// TIA Portal V21 export
FUNCTION "ModeSelect" : Void   // FC7, LAD
{ S7_Optimized_Access := 'TRUE' }
// stored: AutoNumber false, SetENOAutomatically false
BEGIN

REGION Network 1: ****************************MV3000_Enable *****************************
END_REGION

REGION Network 2: "ModeDb".MV3000.Mode.ManualMode.Enable
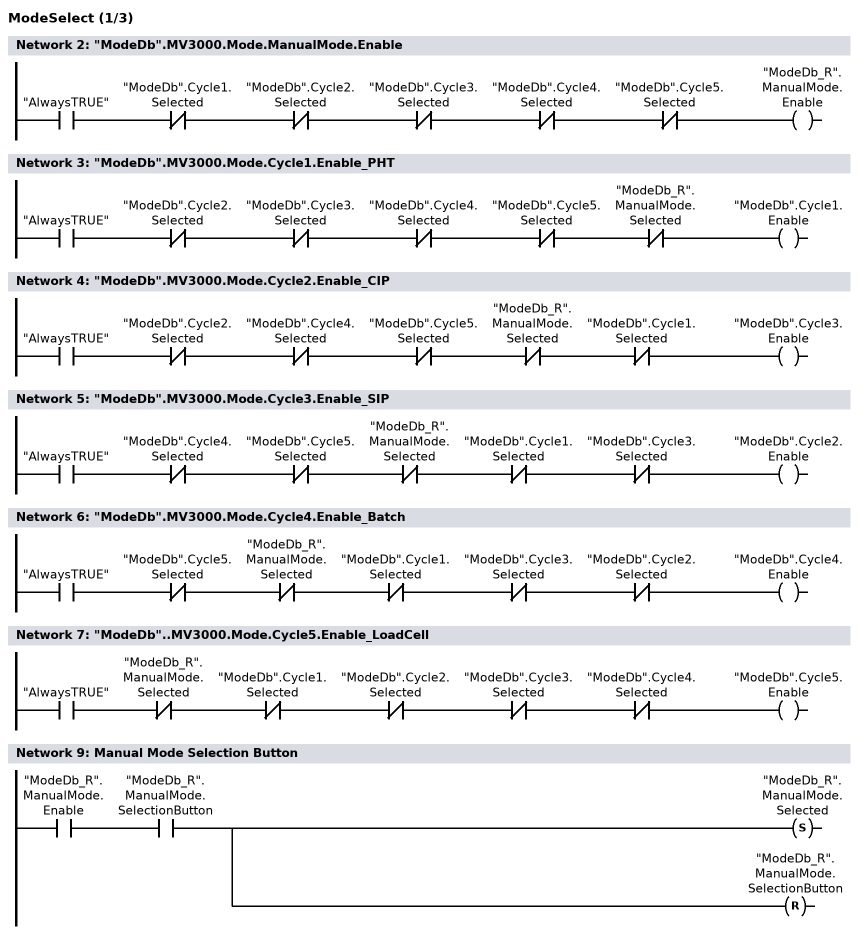
   RUNG wire#powerrail
      Contact( "AlwaysTRUE" )
      I_Contact( "ModeDb".Cycle1.Selected )
      I_Contact( "ModeDb".Cycle2.Selected )
      I_Contact( "ModeDb".Cycle3.Selected )
      I_Contact( "ModeDb".Cycle4.Selected )
      I_Contact( "ModeDb".Cycle5.Selected )
      Coil( "ModeDb_R".ManualMode.Enable )
   END_RUNG
   // the same network as SCL:
   "ModeDb_R".ManualMode.Enable := "AlwaysTRUE" AND NOT "ModeDb".Cycle1.Selected AND NOT "ModeDb".Cycle2.Selected AND NOT "ModeDb".Cycle3.Selected AND NOT "ModeDb".Cycle4.Selected AND NOT "ModeDb".Cycle5.Selected;
END_REGION

REGION Network 3: "ModeDb".MV3000.Mode.Cycle1.Enable_PHT
   RUNG wire#powerrail
      Contact( "AlwaysTRUE" )
      I_Contact( "ModeDb".Cycle2.Selected )
      I_Contact( "ModeDb".Cycle3.Selected )
      I_Contact( "ModeDb".Cycle4.Selected )
      I_Contact( "ModeDb".Cycle5.Selected )
      I_Contact( "ModeDb_R".ManualMode.Selected )
      Coil( "ModeDb".Cycle1.Enable )
   END_RUNG
   // the same network as SCL:
   "ModeDb".Cycle1.Enable := "AlwaysTRUE" AND NOT "ModeDb".Cycle2.Selected AND NOT "ModeDb".Cycle3.Selected AND NOT "ModeDb".Cycle4.Selected AND NOT "ModeDb".Cycle5.Selected AND NOT "ModeDb_R".ManualMode.Selected;
END_REGION

REGION Network 4: "ModeDb".MV3000.Mode.Cycle2.Enable_CIP
   RUNG wire#powerrail
      Contact( "AlwaysTRUE" )
      I_Contact( "ModeDb".Cycle2.Selected )
      I_Contact( "ModeDb".Cycle4.Selected )
      I_Contact( "ModeDb".Cycle5.Selected )
      I_Contact( "ModeDb_R".ManualMode.Selected )
      I_Contact( "ModeDb".Cycle1.Selected )
      Coil( "ModeDb".Cycle3.Enable )
   END_RUNG
   // the same network as SCL:
   "ModeDb".Cycle3.Enable := "AlwaysTRUE" AND NOT "ModeDb".Cycle2.Selected AND NOT "ModeDb".Cycle4.Selected AND NOT "ModeDb".Cycle5.Selected AND NOT "ModeDb_R".ManualMode.Selected AND NOT "ModeDb".Cycle1.Selected;
END_REGION

REGION Network 5: "ModeDb".MV3000.Mode.Cycle3.Enable_SIP
   RUNG wire#powerrail
      Contact( "AlwaysTRUE" )
      I_Contact( "ModeDb".Cycle4.Selected )
      I_Contact( "ModeDb".Cycle5.Selected )
      I_Contact( "ModeDb_R".ManualMode.Selected )
      I_Contact( "ModeDb".Cycle1.Selected )
      I_Contact( "ModeDb".Cycle3.Selected )
      Coil( "ModeDb".Cycle2.Enable )
   END_RUNG
   // the same network as SCL:
   "ModeDb".Cycle2.Enable := "AlwaysTRUE" AND NOT "ModeDb".Cycle4.Selected AND NOT "ModeDb".Cycle5.Selected AND NOT "ModeDb_R".ManualMode.Selected AND NOT "ModeDb".Cycle1.Selected AND NOT "ModeDb".Cycle3.Selected;
END_REGION

REGION Network 6: "ModeDb".MV3000.Mode.Cycle4.Enable_Batch
   RUNG wire#powerrail
      Contact( "AlwaysTRUE" )
      I_Contact( "ModeDb".Cycle5.Selected )
      I_Contact( "ModeDb_R".ManualMode.Selected )
      I_Contact( "ModeDb".Cycle1.Selected )
      I_Contact( "ModeDb".Cycle3.Selected )
      I_Contact( "ModeDb".Cycle2.Selected )
      Coil( "ModeDb".Cycle4.Enable )
   END_RUNG
   // the same network as SCL:
   "ModeDb".Cycle4.Enable := "AlwaysTRUE" AND NOT "ModeDb".Cycle5.Selected AND NOT "ModeDb_R".ManualMode.Selected AND NOT "ModeDb".Cycle1.Selected AND NOT "ModeDb".Cycle3.Selected AND NOT "ModeDb".Cycle2.Selected;
END_REGION

REGION Network 7: "ModeDb"..MV3000.Mode.Cycle5.Enable_LoadCell
   RUNG wire#powerrail
      Contact( "AlwaysTRUE" )
      I_Contact( "ModeDb_R".ManualMode.Selected )
      I_Contact( "ModeDb".Cycle1.Selected )
      I_Contact( "ModeDb".Cycle2.Selected )
      I_Contact( "ModeDb".Cycle3.Selected )
      I_Contact( "ModeDb".Cycle4.Selected )
      Coil( "ModeDb".Cycle5.Enable )
   END_RUNG
   // the same network as SCL:
   "ModeDb".Cycle5.Enable := "AlwaysTRUE" AND NOT "ModeDb_R".ManualMode.Selected AND NOT "ModeDb".Cycle1.Selected AND NOT "ModeDb".Cycle2.Selected AND NOT "ModeDb".Cycle3.Selected AND NOT "ModeDb".Cycle4.Selected;
END_REGION

REGION Network 8: ------------------------------------------------- SELECTION BUTTON -------------------------------------------------
END_REGION

REGION Network 9: Manual Mode Selection Button
   RUNG wire#powerrail
      Contact( "ModeDb_R".ManualMode.Enable )
      Contact( "ModeDb_R".ManualMode.SelectionButton )
      wire#w1
      S_Coil( "ModeDb_R".ManualMode.Selected )
   END_RUNG
   RUNG wire#w1
      R_Coil( "ModeDb_R".ManualMode.SelectionButton )
   END_RUNG
   // the same network as SCL:
   IF "ModeDb_R".ManualMode.Enable AND "ModeDb_R".ManualMode.SelectionButton THEN
       "ModeDb_R".ManualMode.Selected := TRUE;
       "ModeDb_R".ManualMode.SelectionButton := FALSE;
   END_IF;
END_REGION

REGION Network 10: __________________________ VESSEL STATUS__________________________
END_REGION

REGION Network 11: "HmiTags".Cv200VesselStatus
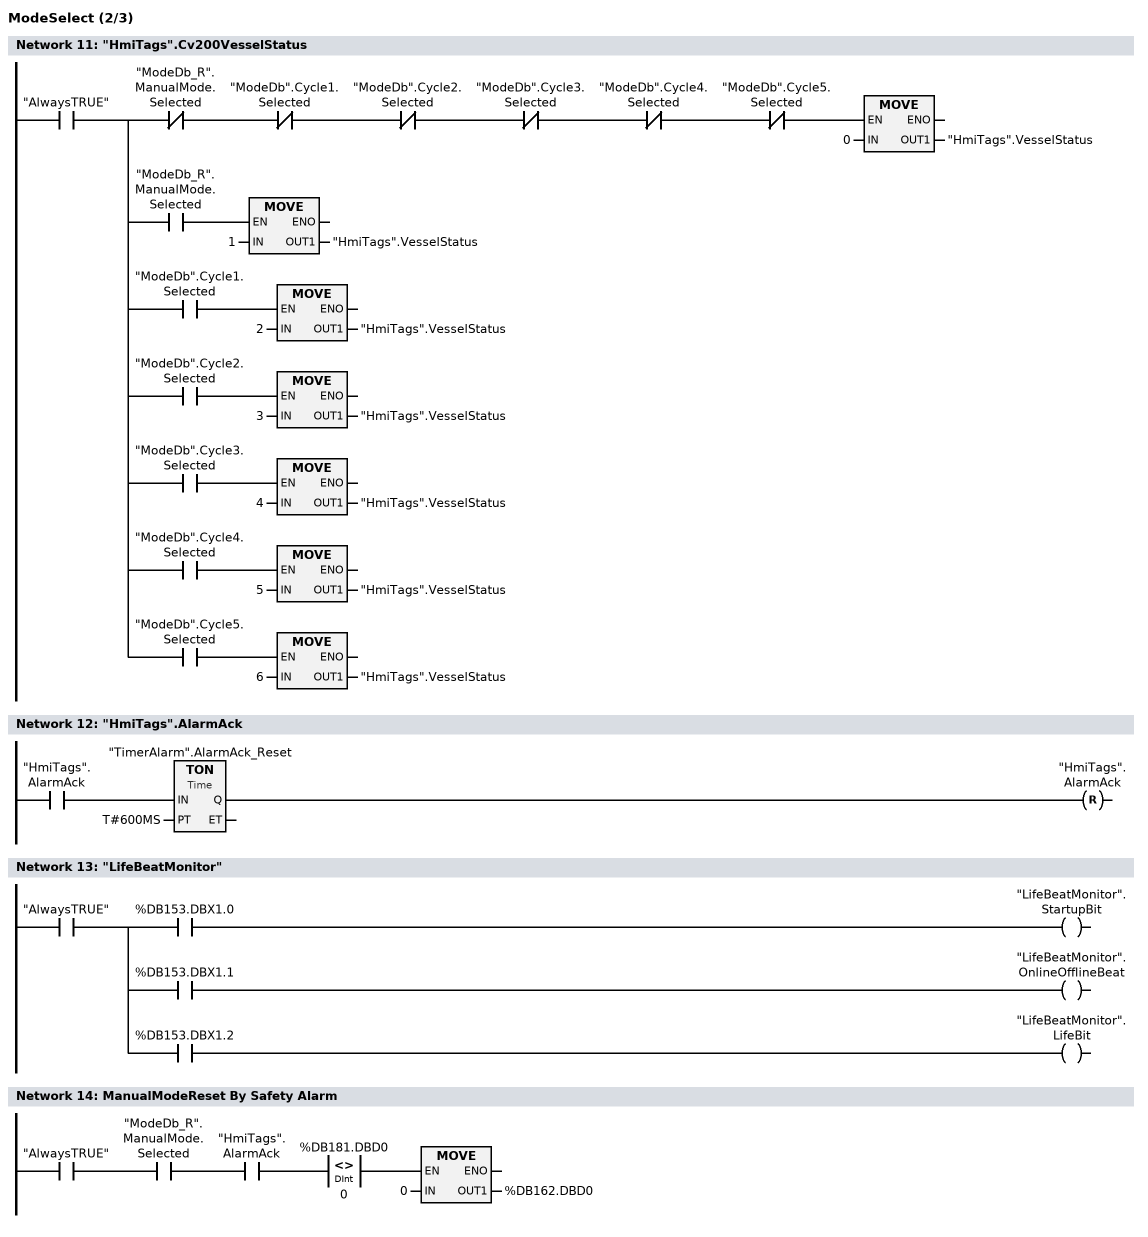
   RUNG wire#powerrail
      Contact( "AlwaysTRUE" )
      wire#w1
      I_Contact( "ModeDb_R".ManualMode.Selected )
      I_Contact( "ModeDb".Cycle1.Selected )
      I_Contact( "ModeDb".Cycle2.Selected )
      I_Contact( "ModeDb".Cycle3.Selected )
      I_Contact( "ModeDb".Cycle4.Selected )
      I_Contact( "ModeDb".Cycle5.Selected )
      Move(in := 0, out1 => "HmiTags".VesselStatus)
   END_RUNG
   RUNG wire#w1
      Contact( "ModeDb_R".ManualMode.Selected )
      Move(in := 1, out1 => "HmiTags".VesselStatus)
   END_RUNG
   RUNG wire#w1
      Contact( "ModeDb".Cycle1.Selected )
      Move(in := 2, out1 => "HmiTags".VesselStatus)
   END_RUNG
   RUNG wire#w1
      Contact( "ModeDb".Cycle2.Selected )
      Move(in := 3, out1 => "HmiTags".VesselStatus)
   END_RUNG
   RUNG wire#w1
      Contact( "ModeDb".Cycle3.Selected )
      Move(in := 4, out1 => "HmiTags".VesselStatus)
   END_RUNG
   RUNG wire#w1
      Contact( "ModeDb".Cycle4.Selected )
      Move(in := 5, out1 => "HmiTags".VesselStatus)
   END_RUNG
   RUNG wire#w1
      Contact( "ModeDb".Cycle5.Selected )
      Move(in := 6, out1 => "HmiTags".VesselStatus)
   END_RUNG
   // the same network as SCL:
   IF "AlwaysTRUE" AND NOT "ModeDb_R".ManualMode.Selected AND NOT "ModeDb".Cycle1.Selected AND NOT "ModeDb".Cycle2.Selected AND NOT "ModeDb".Cycle3.Selected AND NOT "ModeDb".Cycle4.Selected AND NOT "ModeDb".Cycle5.Selected THEN
       "HmiTags".VesselStatus := 0;
   END_IF;
   IF "AlwaysTRUE" AND "ModeDb_R".ManualMode.Selected THEN "HmiTags".VesselStatus := 1; END_IF;
   IF "AlwaysTRUE" AND "ModeDb".Cycle1.Selected THEN "HmiTags".VesselStatus := 2; END_IF;
   IF "AlwaysTRUE" AND "ModeDb".Cycle2.Selected THEN "HmiTags".VesselStatus := 3; END_IF;
   IF "AlwaysTRUE" AND "ModeDb".Cycle3.Selected THEN "HmiTags".VesselStatus := 4; END_IF;
   IF "AlwaysTRUE" AND "ModeDb".Cycle4.Selected THEN "HmiTags".VesselStatus := 5; END_IF;
   IF "AlwaysTRUE" AND "ModeDb".Cycle5.Selected THEN "HmiTags".VesselStatus := 6; END_IF;
END_REGION

REGION Network 12: "HmiTags".AlarmAck
   RUNG wire#powerrail
      Contact( "HmiTags".AlarmAck )
      { S7_Templates := "time_type := Time" } "TimerAlarm".AlarmAck_Reset.TON(pt := T#600MS, et =>)
      R_Coil( "HmiTags".AlarmAck )
   END_RUNG
   // the same network as SCL:
   "TimerAlarm".AlarmAck_Reset.TON(IN := "HmiTags".AlarmAck, PT := T#600MS);
   IF "TimerAlarm".AlarmAck_Reset.Q THEN "HmiTags".AlarmAck := FALSE; END_IF;
END_REGION

REGION Network 13: "LifeBeatMonitor"
   RUNG wire#powerrail
      Contact( "AlwaysTRUE" )
      wire#w1
      Contact( %DB153.DBX1.0 )
      Coil( "LifeBeatMonitor".StartupBit )
   END_RUNG
   RUNG wire#w1
      Contact( %DB153.DBX1.1 )
      Coil( "LifeBeatMonitor".OnlineOfflineBeat )
   END_RUNG
   RUNG wire#w1
      Contact( %DB153.DBX1.2 )
      Coil( "LifeBeatMonitor".LifeBit )
   END_RUNG
   // the same network as SCL:
   "LifeBeatMonitor".StartupBit := "AlwaysTRUE" AND %DB153.DBX1.0;
   "LifeBeatMonitor".OnlineOfflineBeat := "AlwaysTRUE" AND %DB153.DBX1.1;
   "LifeBeatMonitor".LifeBit := "AlwaysTRUE" AND %DB153.DBX1.2;
END_REGION

REGION Network 14: ManualModeReset By Safety Alarm
   RUNG wire#powerrail
      Contact( "AlwaysTRUE" )
      Contact( "ModeDb_R".ManualMode.Selected )
      Contact( "HmiTags".AlarmAck )
      { S7_Templates := "SrcType := DInt" } NE_Contact(in1 := %DB181.DBD0, in2 := 0)
      Move(in := 0, out1 => %DB162.DBD0)
   END_RUNG
   // the same network as SCL:
   IF "AlwaysTRUE" AND "ModeDb_R".ManualMode.Selected AND "HmiTags".AlarmAck AND (%DB181.DBD0 <> 0) THEN
       %DB162.DBD0 := 0;
   END_IF;
END_REGION

REGION Network 15: Master Reset
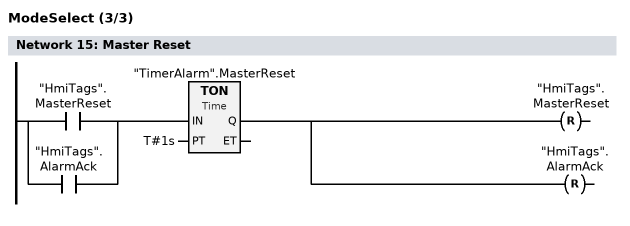
   RUNG wire#powerrail
      Contact( "HmiTags".MasterReset )
      wire#w1
      { S7_Templates := "time_type := Time" } "TimerAlarm".MasterReset.TON(pt := T#1s, et =>)
      wire#w2
      R_Coil( "HmiTags".MasterReset )
   END_RUNG
   RUNG wire#powerrail
      Contact( "HmiTags".AlarmAck )
   END_RUNG wire#w1
   RUNG wire#w2
      R_Coil( "HmiTags".AlarmAck )
   END_RUNG
   // the same network as SCL:
   "TimerAlarm".MasterReset.TON(IN := "HmiTags".MasterReset OR "HmiTags".AlarmAck, PT := T#1s);
   IF "TimerAlarm".MasterReset.Q THEN
       "HmiTags".MasterReset := FALSE;
       "HmiTags".AlarmAck := FALSE;
   END_IF;
END_REGION

REGION Network 16 (SCL): __________________________ Manual Mode Valve REset__________________________
   IF ("ModeDb_R".ManualMode.Abort  = 1 OR "HmiTags".MasterReset = 1) AND "ModeDb_R".ManualMode.Selected = 1 AND
       "ValveDb".Cv01.OpenClose =0 AND
       "ValveDb".Cv02.OpenClose =0 AND
       "ValveDb".Cv03.OpenClose=0  AND
       "ValveDb".Cv04.OpenClose=0 AND
       "ValveDb".Cv05.OpenClose=0 AND
       "ValveDb".Cv06.OpenClose=0 AND
       "ValveDb".Cv07.OpenClose=0 AND
       "ValveDb".Cv08.OpenClose=0 AND
       "ValveDb".Cv09.OpenClose=0 AND
       "ValveDb".Cv10.OpenClose=0 AND
       "ValveDb".Cv11.OpenClose=0 AND
       "ValveDb".Cv12.OpenClose=0 AND
       "ValveDb".Cv13.OpenClose=0 AND
       "ValveDb".Cv14.OpenClose=0 AND
       "ValveDb".Cv15.OpenClose=0 AND
       "ValveDb".Cv16.OpenClose=0 AND
       "ValveDb".Cv17.OpenClose=0 AND
       "ValveDb".Cv18.OpenClose=0 AND
       "ValveDb".Cv19.OpenClose=0 AND
       "ValveDb".Cv20.OpenClose=0 AND
       "ValveDb".Cv21.OpenClose=0 AND
       "ValveDb".Cv22.OpenClose=0 AND
       "ValveDb".Cv23.OpenClose=0 AND
       "ValveDb".Cv24.OpenClose=0 AND
       "ValveDb".Cv25.OpenClose=0 AND
       "ValveDb".Cv26.OpenClose=0 AND
       "ValveDb".Cv27.OpenClose=0 AND
       "ValveDb".Cv28.OpenClose=0 AND
       "ValveDb".Cv29.OpenClose=0 AND
       "ValveDb".Cv30.OpenClose=0 AND
       "ValveDb".Cv31.OpenClose=0 AND
       "ValveDb".Cv32.OpenClose=0 AND
       "ValveDb".Cv33.OpenClose=0 AND
       "ValveDb".Cv34.OpenClose=0 AND
       "ValveDb".Cv35.OpenClose=0 AND
       "ValveDb".Cv36.OpenClose=0 AND
       "ValveDb".Cv37.OpenClose=0 AND
       "ValveDb".Cv38.OpenClose=0 AND
       "ValveDb".Cv39.OpenClose=0 AND  
       "ValveDb".Cv40.OpenClose=0 AND
       "ValveDb".Cv41.OpenClose=0 AND
       "ValveDb".Cv42.OpenClose=0 AND
       "ValveDb".Cv43.OpenClose=0 AND
       "ValveDb".Cv44.OpenClose=0 AND
       "ValveDb".Cv45.OpenClose=0 AND
       "ValveDb".Cv46.OpenClose=0 AND
       "ValveDb".Cv47.OpenClose=0 AND
       "ValveDb".Cv48.OpenClose=0 AND
       "ValveDb".Cv49.OpenClose=0 AND
       "ValveDb".Cv50.OpenClose=0 AND
       "ValveDb".Cv51.OpenClose=0 AND
       "ValveDb".Cv52.OpenClose=0 AND
       "ValveDb".Cv53.OpenClose=0 AND
       "ValveDb".Cv54.OpenClose=0 AND
       "ValveDb".Cv55.OpenClose=0 AND
       "ValveDb".Cv56.OpenClose=0 AND
       "ValveDb".Cv57.OpenClose=0 AND
       "ValveDb".Cv58.OpenClose=0 AND
       "ValveDb".Cv59.OpenClose=0 AND
       "ValveDb".Cv60.OpenClose=0 AND
       "ValveDb".Cv61.OpenClose=0 AND
       "ValveDb".Cv62.OpenClose=0 AND
       "ValveDb".Cv63.OpenClose=0 AND
       "ValveDb".Cv64.OpenClose=0 AND
       "ValveDb".Fbov01.OpenClose=0




   THEN
       "ModeDb_R".ManualMode.Selected := 0 ;
   END_IF;
END_REGION
END_FUNCTION
